TYPE "UDT_Winnc_for_Scada"
VERSION : 0.1
   STRUCT
"Read_write_Symap_Db_Devices_Wincc_Out_module_1_b0_11_Eventsbyte_350_365_b0_1_event_350" :  Bool;
"Read_write_Symap_Db_Devices_Wincc_Out_module_1_b0_11_Eventsbyte_350_365_b0_1_event_351" :  Bool;
"Read_write_Symap_Db_Devices_Wincc_Out_module_1_b0_11_Eventsbyte_350_365_b0_1_event_352" :  Bool;
"Read_write_Symap_Db_Devices_Wincc_Out_module_1_b0_11_Eventsbyte_350_365_b0_1_event_353" :  Bool;
"Read_write_Symap_Db_Devices_Wincc_Out_module_1_b0_11_Eventsbyte_350_365_b0_1_event_354" :  Bool;
"Read_write_Symap_Db_Devices_Wincc_Out_module_1_b0_11_Eventsbyte_350_365_b0_1_event_355" :  Bool;
"Read_write_Symap_Db_Devices_Wincc_Out_module_1_b0_11_Eventsbyte_350_365_b0_1_event_356" :  Bool;
"Read_write_Symap_Db_Devices_Wincc_Out_module_1_b0_11_Eventsbyte_350_365_b0_1_event_357" :  Bool;
"Read_write_Symap_Db_Devices_Wincc_Out_module_1_b0_11_Eventsbyte_350_365_b0_1_event_358" :  Bool;
"Read_write_Symap_Db_Devices_Wincc_Out_module_1_b0_11_Eventsbyte_350_365_b0_1_event_359" :  Bool;
"Read_write_Symap_Db_Devices_Wincc_Out_module_1_b0_11_Eventsbyte_350_365_b0_1_event_360" :  Bool;
"Read_write_Symap_Db_Devices_Wincc_Out_module_1_b0_11_Eventsbyte_350_365_b0_1_event_361" :  Bool;
"Read_write_Symap_Db_Devices_Wincc_Out_module_1_b0_11_Eventsbyte_350_365_b0_1_event_362" :  Bool;
"Read_write_Symap_Db_Devices_Wincc_Out_module_1_b0_11_Eventsbyte_350_365_b0_1_event_363" :  Bool;
"Read_write_Symap_Db_Devices_Wincc_Out_module_1_b0_11_Eventsbyte_350_365_b0_1_event_364" :  Bool;
"Read_write_Symap_Db_Devices_Wincc_Out_module_1_b0_11_Eventsbyte_350_365_b0_1_event_365" :  Bool;
"Read_write_Symap_Db_Devices_Wincc_Out_module_1_b0_11_Control_Byte_b2_3_Change_work" :  Bool;
"Read_write_Symap_Db_Devices_Wincc_Out_module_1_b0_11_Control_Byte_b2_3_Res" :  Bool;
"Read_write_Symap_Db_Devices_Wincc_Out_module_1_b0_11_Control_Byte_b2_3_Set_time" :  Bool;
"Read_write_Symap_Db_Devices_Wincc_Out_module_1_b0_11_Control_Byte_b2_3_Cb3" :  Bool;
"Read_write_Symap_Db_Devices_Wincc_Out_module_1_b0_11_Control_Byte_b2_3_Cb4" :  Bool;
"Read_write_Symap_Db_Devices_Wincc_Out_module_1_b0_11_Control_Byte_b2_3_Cb5" :  Bool;
"Read_write_Symap_Db_Devices_Wincc_Out_module_1_b0_11_Control_Byte_b2_3_Cb6" :  Bool;
"Read_write_Symap_Db_Devices_Wincc_Out_module_1_b0_11_Control_Byte_b2_3_Cb7" :  Bool;
"Read_write_Symap_Db_Devices_Wincc_Out_module_1_b0_11_Control_Byte_b2_3_local" :  Bool;
"Read_write_Symap_Db_Devices_Wincc_Out_module_1_b0_11_Control_Byte_b2_3_remote" :  Bool;
"Read_write_Symap_Db_Devices_Wincc_Out_module_1_b0_11_Control_Byte_b2_3_SCADA" :  Bool;
"Read_write_Symap_Db_Devices_Wincc_Out_module_1_b0_11_Control_Byte_b2_3_test_local" :  Bool;
"Read_write_Symap_Db_Devices_Wincc_Out_module_1_b0_11_Control_Byte_b2_3_test_remote" :  Bool;
"Read_write_Symap_Db_Devices_Wincc_Out_module_1_b0_11_Control_Byte_b2_3_NM5" :  Bool;
"Read_write_Symap_Db_Devices_Wincc_Out_module_1_b0_11_Control_Byte_b2_3_NM6" :  Bool;
"Read_write_Symap_Db_Devices_Wincc_Out_module_1_b0_11_Control_Byte_b2_3_NM7" :  Bool;
"Read_write_Symap_Db_Devices_Wincc_Out_module_1_b0_11_Time_set_b4_11_month" :  Byte;
"Read_write_Symap_Db_Devices_Wincc_Out_module_1_b0_11_Time_set_b4_11_year" :  Byte;
"Read_write_Symap_Db_Devices_Wincc_Out_module_1_b0_11_Time_set_b4_11_hour" :  Byte;
"Read_write_Symap_Db_Devices_Wincc_Out_module_1_b0_11_Time_set_b4_11_day" :  Byte;
"Read_write_Symap_Db_Devices_Wincc_Out_module_1_b0_11_Time_set_b4_11_second" :  Byte;
"Read_write_Symap_Db_Devices_Wincc_Out_module_1_b0_11_Time_set_b4_11_minute" :  Byte;
"Read_write_Symap_Db_Devices_Wincc_Out_module_1_b0_11_Time_set_b4_11_millisecondhigh_Byte" :  Byte;
"Read_write_Symap_Db_Devices_Wincc_Out_module_1_b0_11_Time_set_b4_11_millisecondlow_Byte" :  Byte;
"Read_write_Symap_Db_Devices_Wincc_Out_module_30_b12_15_instr_No_1_b5" :  Byte;
"Read_write_Symap_Db_Devices_Wincc_Out_module_30_b12_15_instr_No_2_b6" :  Byte;
"Read_write_Symap_Db_Devices_Wincc_Out_module_30_b12_15_Data_val_1_b7" :  Byte;
"Read_write_Symap_Db_Devices_Wincc_Out_module_30_b12_15_Data_val_2_b8" :  Byte;
"Read_write_Symap_Db_Devices_Wincc_Filtered_FDR_FR_b14_15" :  Real;
"Read_write_Symap_Db_Devices_Wincc_Filtered_FDR_U1_b16_17" :  Real;
"Read_write_Symap_Db_Devices_Wincc_Filtered_FDR_U2_b18_19" :  Real;
"Read_write_Symap_Db_Devices_Wincc_Filtered_FDR_U3_b20_21" :  Real;
"Read_write_Symap_Db_Devices_Wincc_Filtered_FDR_U12_b22_23" :  Real;
"Read_write_Symap_Db_Devices_Wincc_Filtered_FDR_U13_b24_25" :  Real;
"Read_write_Symap_Db_Devices_Wincc_Filtered_FDR_U23_b26_27" :  Real;
"Read_write_Symap_Db_Devices_Wincc_Filtered_FDR_UAvr_b28_29" :  Real;
"Read_write_Symap_Db_Devices_Wincc_Filtered_BUS1_FR_b31_32" :  Real;
"Read_write_Symap_Db_Devices_Wincc_Filtered_BUS1_U1_b32_33" :  Real;
"Read_write_Symap_Db_Devices_Wincc_Filtered_BUS1_U2_b34_35" :  Real;
"Read_write_Symap_Db_Devices_Wincc_Filtered_BUS1_U3_b36_37" :  Real;
"Read_write_Symap_Db_Devices_Wincc_Filtered_BUS1_U12_b38_39" :  Real;
"Read_write_Symap_Db_Devices_Wincc_Filtered_BUS1_U13_b40_41" :  Real;
"Read_write_Symap_Db_Devices_Wincc_Filtered_BUS1_U23_b42_43" :  Real;
"Read_write_Symap_Db_Devices_Wincc_Filtered_BUS1_UAvr_b44_45" :  Real;
"Read_write_Symap_Db_Devices_Wincc_Filtered_BUS2_FR_b46_47" :  Real;
"Read_write_Symap_Db_Devices_Wincc_Filtered_BUS2_U1_b48_49" :  Real;
"Read_write_Symap_Db_Devices_Wincc_Filtered_BUS2_U2_b50_51" :  Real;
"Read_write_Symap_Db_Devices_Wincc_Filtered_BUS2_U3_b52_53" :  Real;
"Read_write_Symap_Db_Devices_Wincc_Filtered_BUS2_U12_b54_55" :  Real;
"Read_write_Symap_Db_Devices_Wincc_Filtered_BUS2_U13_b56_57" :  Real;
"Read_write_Symap_Db_Devices_Wincc_Filtered_BUS2_U23_b58_59" :  Real;
"Read_write_Symap_Db_Devices_Wincc_Filtered_BUS2_UAvr_b60_61" :  Real;
"Read_write_Symap_Db_Devices_Wincc_Filtered_FDR_I1_b62_63" :  Real;
"Read_write_Symap_Db_Devices_Wincc_Filtered_FDR_I2_b64_65" :  Real;
"Read_write_Symap_Db_Devices_Wincc_Filtered_FDR_I3_b65_67" :  Real;
"Read_write_Symap_Db_Devices_Wincc_Filtered_FDR_IAvr_b68_69" :  Real;
"Read_write_Symap_Db_Devices_Wincc_Filtered_FDR_P" :  Real;
"Read_write_Symap_Db_Devices_Wincc_Filtered_FDR_Q" :  Real;
"Read_write_Symap_Db_Devices_Wincc_Filtered_FDR_S" :  Real;
"Read_write_Symap_Db_Devices_Wincc_Filtered_FDR_PF" :  Real;
"Read_write_Symap_Db_Devices_Wincc_Filtered_FDR_PL1" :  Real;
"Read_write_Symap_Db_Devices_Wincc_Filtered_FDR_PL2" :  Real;
"Read_write_Symap_Db_Devices_Wincc_Filtered_FDR_PL3" :  Real;
"Read_write_Symap_Db_Devices_Wincc_Filtered_FDR_QL1" :  Real;
"Read_write_Symap_Db_Devices_Wincc_Filtered_FDR_QL2" :  Real;
"Read_write_Symap_Db_Devices_Wincc_Filtered_FDR_QL3" :  Real;
"Read_write_Symap_Db_Devices_Wincc_Filtered_FDR_PFL1" :  Real;
"Read_write_Symap_Db_Devices_Wincc_Filtered_FDR_PFL2" :  Real;
"Read_write_Symap_Db_Devices_Wincc_Filtered_FDR_PFL3" :  Real;
"Read_write_Symap_Db_Devices_Wincc_Factor_modul_7_b14_29_Fc_FDR_FR_b14_15" :  Real;
"Read_write_Symap_Db_Devices_Wincc_Factor_modul_7_b14_29_Fc_FDR_U1_b16_17" :  Real;
"Read_write_Symap_Db_Devices_Wincc_Factor_modul_7_b14_29_Fc_FDR_U2_b18_19" :  Real;
"Read_write_Symap_Db_Devices_Wincc_Factor_modul_7_b14_29_Fc_FDR_U3_b20_21" :  Real;
"Read_write_Symap_Db_Devices_Wincc_Factor_modul_7_b14_29_Fc_FDR_U12_b22_23" :  Real;
"Read_write_Symap_Db_Devices_Wincc_Factor_modul_7_b14_29_Fc_FDR_U13_b24_25" :  Real;
"Read_write_Symap_Db_Devices_Wincc_Factor_modul_7_b14_29_Fc_FDR_U23_b26_27" :  Real;
"Read_write_Symap_Db_Devices_Wincc_Factor_modul_7_b14_29_Fc_FDR_UAvr_b28_29" :  Real;
"Read_write_Symap_Db_Devices_Wincc_Factor_modul_830_45_Fc_BUS1_FR_b31_32" :  Real;
"Read_write_Symap_Db_Devices_Wincc_Factor_modul_830_45_Fc_BUS1_U1_b32_33" :  Real;
"Read_write_Symap_Db_Devices_Wincc_Factor_modul_830_45_Fc_BUS1_U2_b34_35" :  Real;
"Read_write_Symap_Db_Devices_Wincc_Factor_modul_830_45_Fc_BUS1_U3_b36_37" :  Real;
"Read_write_Symap_Db_Devices_Wincc_Factor_modul_830_45_Fc_BUS1_U12_b38_39" :  Real;
"Read_write_Symap_Db_Devices_Wincc_Factor_modul_830_45_Fc_BUS1_U13_b40_41" :  Real;
"Read_write_Symap_Db_Devices_Wincc_Factor_modul_830_45_Fc_BUS1_U23_b42_43" :  Real;
"Read_write_Symap_Db_Devices_Wincc_Factor_modul_830_45_Fc_BUS1_UAvr_b44_45" :  Real;
"Read_write_Symap_Db_Devices_Wincc_Factor_modul_9_b46_61_Fc_BUS2_FR_b46_47" :  Real;
"Read_write_Symap_Db_Devices_Wincc_Factor_modul_9_b46_61_Fc_BUS2_U1_b48_49" :  Real;
"Read_write_Symap_Db_Devices_Wincc_Factor_modul_9_b46_61_Fc_BUS2_U2_b50_51" :  Real;
"Read_write_Symap_Db_Devices_Wincc_Factor_modul_9_b46_61_Fc_BUS2_U3_b52_53" :  Real;
"Read_write_Symap_Db_Devices_Wincc_Factor_modul_9_b46_61_Fc_BUS2_U12_b54_55" :  Real;
"Read_write_Symap_Db_Devices_Wincc_Factor_modul_9_b46_61_Fc_BUS2_U13_b56_57" :  Real;
"Read_write_Symap_Db_Devices_Wincc_Factor_modul_9_b46_61_Fc_BUS2_U23_b58_59" :  Real;
"Read_write_Symap_Db_Devices_Wincc_Factor_modul_9_b46_61_Fc_BUS2_UAvr_b60_61" :  Real;
"Read_write_Symap_Db_Devices_Wincc_Factor_modul_10_b62_69_Fc_FDR_I1_b62_63" :  Real;
"Read_write_Symap_Db_Devices_Wincc_Factor_modul_10_b62_69_Fc_FDR_I2_b64_65" :  Real;
"Read_write_Symap_Db_Devices_Wincc_Factor_modul_10_b62_69_Fc_FDR_I3_b65_67" :  Real;
"Read_write_Symap_Db_Devices_Wincc_Factor_modul_10_b62_69_Fc_FDR_IAvr_b68_69" :  Real;
"Read_write_Symap_Db_Devices_Wincc_Factor_modul_12_b70_77_Fc_FDR_P_b70_71" :  Real;
"Read_write_Symap_Db_Devices_Wincc_Factor_modul_12_b70_77_Fc_FDR_Q_b72_73" :  Real;
"Read_write_Symap_Db_Devices_Wincc_Factor_modul_12_b70_77_Fc_FDR_S_b74_75" :  Real;
"Read_write_Symap_Db_Devices_Wincc_Factor_modul_12_b70_77_Fc_FDR_PF_b76_77" :  Real;
"Read_write_Symap_Db_Devices_Wincc_Factor_modul_13_b78_83_Fc_FDR_PL1_b78_79" :  Real;
"Read_write_Symap_Db_Devices_Wincc_Factor_modul_13_b78_83_Fc_FDR_PL2_b80_81" :  Real;
"Read_write_Symap_Db_Devices_Wincc_Factor_modul_13_b78_83_Fc_FDR_PL3_b82_83" :  Real;
"Read_write_Symap_Db_Devices_Wincc_Factor_modul_14_b84_89_Fc_FDR_QL1_b84_85" :  Real;
"Read_write_Symap_Db_Devices_Wincc_Factor_modul_14_b84_89_Fc_FDR_QL2_b86_87" :  Real;
"Read_write_Symap_Db_Devices_Wincc_Factor_modul_14_b84_89_Fc_FDR_QL3_b88_89" :  Real;
"Read_write_Symap_Db_Devices_Wincc_Factor_modul_15_b90_95_Fc_FDR_PFL1_b90_91" :  Real;
"Read_write_Symap_Db_Devices_Wincc_Factor_modul_15_b90_95_Fc_FDR_PFL2_b92_93" :  Real;
"Read_write_Symap_Db_Devices_Wincc_Factor_modul_15_b90_95_Fc_FDR_PFL3_b94_95" :  Real;
"Read_write_Symap_Db_Devices_Wincc_Factor_modul_18_b96_111_Fc_P_activ_b96_99" :  Real;
"Read_write_Symap_Db_Devices_Wincc_Factor_modul_18_b96_111_Fc_P_obr_b100_103" :  Real;
"Read_write_Symap_Db_Devices_Wincc_Factor_modul_18_b96_111_Fc_P_emk_reakt_b104_107" :  Real;
"Read_write_Symap_Db_Devices_Wincc_Factor_modul_18_b96_111_Fc_P_ind_reakt_b108_111" :  Real;
"Read_write_Symap_Db_Devices_Wincc_Factor_modul_16_b112_119_Fc_Io1_b112_113" :  Real;
"Read_write_Symap_Db_Devices_Wincc_Factor_modul_16_b112_119_Fc_Uo1_b114_115" :  Real;
"Read_write_Symap_Db_Devices_Wincc_Factor_modul_16_b112_119_Fc_Po1_b116_117" :  Real;
"Read_write_Symap_Db_Devices_Wincc_Factor_modul_16_b112_119_Fc_Qo1_b118_119" :  Real;
"Read_write_Symap_Db_Devices_Wincc_Factor_modul_25_b120_129_Fc_Alarm1_b120_121" :  Real;
"Read_write_Symap_Db_Devices_Wincc_Factor_modul_25_b120_129_Fc_Alarm2_b122_123" :  Real;
"Read_write_Symap_Db_Devices_Wincc_Factor_modul_25_b120_129_Fc_Alarm3_b124_125" :  Real;
"Read_write_Symap_Db_Devices_Wincc_Factor_modul_25_b120_129_Fc_Alarm4_b126_127" :  Real;
"Read_write_Symap_Db_Devices_Wincc_Factor_modul_25_b120_129_Fc_Alarm5_b128_129" :  Real;
"Read_write_Symap_Db_Devices_Wincc_Factor_modul_31_b130_155_Fc_PM_Gen_number_b130_131" :  Real;
"Read_write_Symap_Db_Devices_Wincc_Factor_modul_31_b130_155_Fc_PM_BCG_prstatus_b132_133" :  Real;
"Read_write_Symap_Db_Devices_Wincc_Factor_modul_31_b130_155_Fc_PM_BCG_ownstatus_b134_135" :  Real;
"Read_write_Symap_Db_Devices_Wincc_Factor_modul_31_b130_155_Fc_PM_BCG_netstatus_b136_137" :  Real;
"Read_write_Symap_Db_Devices_Wincc_Factor_modul_31_b130_155_Fc_PM_8_9_b138_139" :  Real;
"Read_write_Symap_Db_Devices_Wincc_Factor_modul_31_b130_155_Fc_PM_10_11_b140_141" :  Real;
"Read_write_Symap_Db_Devices_Wincc_Factor_modul_31_b130_155_Fc_PM_12_13_b142_143" :  Real;
"Read_write_Symap_Db_Devices_Wincc_Factor_modul_31_b130_155_Fc_PM_14_15_b144_145" :  Real;
"Read_write_Symap_Db_Devices_Wincc_Factor_modul_31_b130_155_Fc_PM_16_17_b146_147" :  Real;
"Read_write_Symap_Db_Devices_Wincc_Factor_modul_31_b130_155_Fc_PM_18_19_b148_149" :  Real;
"Read_write_Symap_Db_Devices_Wincc_Factor_modul_31_b130_155_Fc_PM_20_21_b150_151" :  Real;
"Read_write_Symap_Db_Devices_Wincc_Factor_modul_31_b130_155_Fc_PM_asym_load_point_b152_153" :  Real;
"Read_write_Symap_Db_Devices_Wincc_Factor_modul_31_b130_155_Fc_PM_asym_power_factor_b151_155" :  Real;
"Read_write_Symap_Db_Devices_Wincc_Factor_modul_32_b156_173_Fc_P_kw_b156_157" :  Real;
"Read_write_Symap_Db_Devices_Wincc_Factor_modul_32_b156_173_Fc_P_ps_b158_159" :  Real;
"Read_write_Symap_Db_Devices_Wincc_Factor_modul_32_b156_173_Fc_F_I_amp_b160_161" :  Real;
"Read_write_Symap_Db_Devices_Wincc_Factor_modul_32_b156_173_Fc_F_I_ps_b162_163" :  Real;
"Read_write_Symap_Db_Devices_Wincc_Factor_modul_32_b156_173_Fc_F_U_b164_165" :  Real;
"Read_write_Symap_Db_Devices_Wincc_Factor_modul_32_b156_173_Fc_F_freg_b166_167" :  Real;
"Read_write_Symap_Db_Devices_Wincc_Factor_modul_32_b156_173_Fc_F_cosf_b168_169" :  Real;
"Read_write_Symap_Db_Devices_Wincc_Factor_modul_32_b156_173_Fc_B1_U_b170_171" :  Real;
"Read_write_Symap_Db_Devices_Wincc_Factor_modul_32_b156_173_Fc_B1_freg1_b172_173" :  Real;
"Read_write_Symap_Db_Devices_Wincc_Factor_modul_33_b174_189_Fc_RPM_b174_175" :  Real;
"Read_write_Symap_Db_Devices_Wincc_Factor_modul_33_b174_189_Fc_BR1_ON_cycles_b176_177" :  Real;
"Read_write_Symap_Db_Devices_Wincc_Factor_modul_33_b174_189_Fc_BR2_ON_cycles_b178_179" :  Real;
"Read_write_Symap_Db_Devices_Wincc_Factor_modul_33_b174_189_Fc_BR3_ON_cycles_b180_181" :  Real;
"Read_write_Symap_Db_Devices_Wincc_Factor_modul_33_b174_189_Fc_Start_counter_b182_183" :  Real;
"Read_write_Symap_Db_Devices_Wincc_Factor_modul_33_b174_189_Fc_DP_MD33_R1_b184_185" :  Real;
"Read_write_Symap_Db_Devices_Wincc_Factor_modul_33_b174_189_Fc_DP_MD33_R2_b186_187" :  Real;
"Read_write_Symap_Db_Devices_Wincc_Factor_modul_33_b174_189_Fc_DP_MD33_R3_b188_189" :  Real;
"Read_write_Symap_Db_Devices_Wincc_K_Filter_modul_7_b14_29_Fc_FDR_FR_b14_15" :  Real;
"Read_write_Symap_Db_Devices_Wincc_K_Filter_modul_7_b14_29_Fc_FDR_U1_b16_17" :  Real;
"Read_write_Symap_Db_Devices_Wincc_K_Filter_modul_7_b14_29_Fc_FDR_U2_b18_19" :  Real;
"Read_write_Symap_Db_Devices_Wincc_K_Filter_modul_7_b14_29_Fc_FDR_U3_b20_21" :  Real;
"Read_write_Symap_Db_Devices_Wincc_K_Filter_modul_7_b14_29_Fc_FDR_U12_b22_23" :  Real;
"Read_write_Symap_Db_Devices_Wincc_K_Filter_modul_7_b14_29_Fc_FDR_U13_b24_25" :  Real;
"Read_write_Symap_Db_Devices_Wincc_K_Filter_modul_7_b14_29_Fc_FDR_U23_b26_27" :  Real;
"Read_write_Symap_Db_Devices_Wincc_K_Filter_modul_7_b14_29_Fc_FDR_UAvr_b28_29" :  Real;
"Read_write_Symap_Db_Devices_Wincc_K_Filter_modul_830_45_Fc_BUS1_FR_b31_32" :  Real;
"Read_write_Symap_Db_Devices_Wincc_K_Filter_modul_830_45_Fc_BUS1_U1_b32_33" :  Real;
"Read_write_Symap_Db_Devices_Wincc_K_Filter_modul_830_45_Fc_BUS1_U2_b34_35" :  Real;
"Read_write_Symap_Db_Devices_Wincc_K_Filter_modul_830_45_Fc_BUS1_U3_b36_37" :  Real;
"Read_write_Symap_Db_Devices_Wincc_K_Filter_modul_830_45_Fc_BUS1_U12_b38_39" :  Real;
"Read_write_Symap_Db_Devices_Wincc_K_Filter_modul_830_45_Fc_BUS1_U13_b40_41" :  Real;
"Read_write_Symap_Db_Devices_Wincc_K_Filter_modul_830_45_Fc_BUS1_U23_b42_43" :  Real;
"Read_write_Symap_Db_Devices_Wincc_K_Filter_modul_830_45_Fc_BUS1_UAvr_b44_45" :  Real;
"Read_write_Symap_Db_Devices_Wincc_K_Filter_modul_9_b46_61_Fc_BUS2_FR_b46_47" :  Real;
"Read_write_Symap_Db_Devices_Wincc_K_Filter_modul_9_b46_61_Fc_BUS2_U1_b48_49" :  Real;
"Read_write_Symap_Db_Devices_Wincc_K_Filter_modul_9_b46_61_Fc_BUS2_U2_b50_51" :  Real;
"Read_write_Symap_Db_Devices_Wincc_K_Filter_modul_9_b46_61_Fc_BUS2_U3_b52_53" :  Real;
"Read_write_Symap_Db_Devices_Wincc_K_Filter_modul_9_b46_61_Fc_BUS2_U12_b54_55" :  Real;
"Read_write_Symap_Db_Devices_Wincc_K_Filter_modul_9_b46_61_Fc_BUS2_U13_b56_57" :  Real;
"Read_write_Symap_Db_Devices_Wincc_K_Filter_modul_9_b46_61_Fc_BUS2_U23_b58_59" :  Real;
"Read_write_Symap_Db_Devices_Wincc_K_Filter_modul_9_b46_61_Fc_BUS2_UAvr_b60_61" :  Real;
"Read_write_Symap_Db_Devices_Wincc_K_Filter_modul_10_b62_69_Fc_FDR_I1_b62_63" :  Real;
"Read_write_Symap_Db_Devices_Wincc_K_Filter_modul_10_b62_69_Fc_FDR_I2_b64_65" :  Real;
"Read_write_Symap_Db_Devices_Wincc_K_Filter_modul_10_b62_69_Fc_FDR_I3_b65_67" :  Real;
"Read_write_Symap_Db_Devices_Wincc_K_Filter_modul_10_b62_69_Fc_FDR_IAvr_b68_69" :  Real;
"Read_write_Symap_Db_Devices_Wincc_K_Filter_modul_12_b70_77_Fc_FDR_P_b70_71" :  Real;
"Read_write_Symap_Db_Devices_Wincc_K_Filter_modul_12_b70_77_Fc_FDR_Q_b72_73" :  Real;
"Read_write_Symap_Db_Devices_Wincc_K_Filter_modul_12_b70_77_Fc_FDR_S_b74_75" :  Real;
"Read_write_Symap_Db_Devices_Wincc_K_Filter_modul_12_b70_77_Fc_FDR_PF_b76_77" :  Real;
"Read_write_Symap_Db_Devices_Wincc_K_Filter_modul_13_b78_83_Fc_FDR_PL1_b78_79" :  Real;
"Read_write_Symap_Db_Devices_Wincc_K_Filter_modul_13_b78_83_Fc_FDR_PL2_b80_81" :  Real;
"Read_write_Symap_Db_Devices_Wincc_K_Filter_modul_13_b78_83_Fc_FDR_PL3_b82_83" :  Real;
"Read_write_Symap_Db_Devices_Wincc_K_Filter_modul_14_b84_89_Fc_FDR_QL1_b84_85" :  Real;
"Read_write_Symap_Db_Devices_Wincc_K_Filter_modul_14_b84_89_Fc_FDR_QL2_b86_87" :  Real;
"Read_write_Symap_Db_Devices_Wincc_K_Filter_modul_14_b84_89_Fc_FDR_QL3_b88_89" :  Real;
"Read_write_Symap_Db_Devices_Wincc_K_Filter_modul_15_b90_95_Fc_FDR_PFL1_b90_91" :  Real;
"Read_write_Symap_Db_Devices_Wincc_K_Filter_modul_15_b90_95_Fc_FDR_PFL2_b92_93" :  Real;
"Read_write_Symap_Db_Devices_Wincc_K_Filter_modul_15_b90_95_Fc_FDR_PFL3_b94_95" :  Real;
"Read_write_Symap_Db_Devices_Wincc_K_Filter_modul_18_b96_111_Fc_P_activ_b96_99" :  Real;
"Read_write_Symap_Db_Devices_Wincc_K_Filter_modul_18_b96_111_Fc_P_obr_b100_103" :  Real;
"Read_write_Symap_Db_Devices_Wincc_K_Filter_modul_18_b96_111_Fc_P_emk_reakt_b104_107" :  Real;
"Read_write_Symap_Db_Devices_Wincc_K_Filter_modul_18_b96_111_Fc_P_ind_reakt_b108_111" :  Real;
"Read_write_Symap_Db_Devices_Wincc_K_Filter_modul_16_b112_119_Fc_Io1_b112_113" :  Real;
"Read_write_Symap_Db_Devices_Wincc_K_Filter_modul_16_b112_119_Fc_Uo1_b114_115" :  Real;
"Read_write_Symap_Db_Devices_Wincc_K_Filter_modul_16_b112_119_Fc_Po1_b116_117" :  Real;
"Read_write_Symap_Db_Devices_Wincc_K_Filter_modul_16_b112_119_Fc_Qo1_b118_119" :  Real;
"Read_write_Symap_Db_Devices_Wincc_K_Filter_modul_25_b120_129_Fc_Alarm1_b120_121" :  Real;
"Read_write_Symap_Db_Devices_Wincc_K_Filter_modul_25_b120_129_Fc_Alarm2_b122_123" :  Real;
"Read_write_Symap_Db_Devices_Wincc_K_Filter_modul_25_b120_129_Fc_Alarm3_b124_125" :  Real;
"Read_write_Symap_Db_Devices_Wincc_K_Filter_modul_25_b120_129_Fc_Alarm4_b126_127" :  Real;
"Read_write_Symap_Db_Devices_Wincc_K_Filter_modul_25_b120_129_Fc_Alarm5_b128_129" :  Real;
"Read_write_Symap_Db_Devices_Wincc_K_Filter_modul_31_b130_155_Fc_PM_Gen_number_b130_131" :  Real;
"Read_write_Symap_Db_Devices_Wincc_K_Filter_modul_31_b130_155_Fc_PM_BCG_prstatus_b132_133" :  Real;
"Read_write_Symap_Db_Devices_Wincc_K_Filter_modul_31_b130_155_Fc_PM_BCG_ownstatus_b134_135" :  Real;
"Read_write_Symap_Db_Devices_Wincc_K_Filter_modul_31_b130_155_Fc_PM_BCG_netstatus_b136_137" :  Real;
"Read_write_Symap_Db_Devices_Wincc_K_Filter_modul_31_b130_155_Fc_PM_8_9_b138_139" :  Real;
"Read_write_Symap_Db_Devices_Wincc_K_Filter_modul_31_b130_155_Fc_PM_10_11_b140_141" :  Real;
"Read_write_Symap_Db_Devices_Wincc_K_Filter_modul_31_b130_155_Fc_PM_12_13_b142_143" :  Real;
"Read_write_Symap_Db_Devices_Wincc_K_Filter_modul_31_b130_155_Fc_PM_14_15_b144_145" :  Real;
"Read_write_Symap_Db_Devices_Wincc_K_Filter_modul_31_b130_155_Fc_PM_16_17_b146_147" :  Real;
"Read_write_Symap_Db_Devices_Wincc_K_Filter_modul_31_b130_155_Fc_PM_18_19_b148_149" :  Real;
"Read_write_Symap_Db_Devices_Wincc_K_Filter_modul_31_b130_155_Fc_PM_20_21_b150_151" :  Real;
"Read_write_Symap_Db_Devices_Wincc_K_Filter_modul_31_b130_155_Fc_PM_asym_load_point_b152_153" :  Real;
"Read_write_Symap_Db_Devices_Wincc_K_Filter_modul_31_b130_155_Fc_PM_asym_power_factor_b151_155" :  Real;
"Read_write_Symap_Db_Devices_Wincc_K_Filter_modul_32_b156_173_Fc_P_kw_b156_157" :  Real;
"Read_write_Symap_Db_Devices_Wincc_K_Filter_modul_32_b156_173_Fc_P_ps_b158_159" :  Real;
"Read_write_Symap_Db_Devices_Wincc_K_Filter_modul_32_b156_173_Fc_F_I_amp_b160_161" :  Real;
"Read_write_Symap_Db_Devices_Wincc_K_Filter_modul_32_b156_173_Fc_F_I_ps_b162_163" :  Real;
"Read_write_Symap_Db_Devices_Wincc_K_Filter_modul_32_b156_173_Fc_F_U_b164_165" :  Real;
"Read_write_Symap_Db_Devices_Wincc_K_Filter_modul_32_b156_173_Fc_F_freg_b166_167" :  Real;
"Read_write_Symap_Db_Devices_Wincc_K_Filter_modul_32_b156_173_Fc_F_cosf_b168_169" :  Real;
"Read_write_Symap_Db_Devices_Wincc_K_Filter_modul_32_b156_173_Fc_B1_U_b170_171" :  Real;
"Read_write_Symap_Db_Devices_Wincc_K_Filter_modul_32_b156_173_Fc_B1_freg1_b172_173" :  Real;
"Read_write_Symap_Db_Devices_Wincc_K_Filter_modul_33_b174_189_Fc_RPM_b174_175" :  Real;
"Read_write_Symap_Db_Devices_Wincc_K_Filter_modul_33_b174_189_Fc_BR1_ON_cycles_b176_177" :  Real;
"Read_write_Symap_Db_Devices_Wincc_K_Filter_modul_33_b174_189_Fc_BR2_ON_cycles_b178_179" :  Real;
"Read_write_Symap_Db_Devices_Wincc_K_Filter_modul_33_b174_189_Fc_BR3_ON_cycles_b180_181" :  Real;
"Read_write_Symap_Db_Devices_Wincc_K_Filter_modul_33_b174_189_Fc_Start_counter_b182_183" :  Real;
"Read_write_Symap_Db_Devices_Wincc_K_Filter_modul_33_b174_189_Fc_DP_MD33_R1_b184_185" :  Real;
"Read_write_Symap_Db_Devices_Wincc_K_Filter_modul_33_b174_189_Fc_DP_MD33_R2_b186_187" :  Real;
"Read_write_Symap_Db_Devices_Wincc_K_Filter_modul_33_b174_189_Fc_DP_MD33_R3_b188_189" :  Real;
   END_STRUCT;

END_TYPE

